Fanuc KAREL source: kt00120.KL

-- PROVISIONAL review KL for V770-1; original PC SHA256 89c0cbe0fdb6aaab56bf269acc3bfb9269b738d73fb216a7128dd25fbaf1ecd8
-- Incomplete behavior may be omitted. Consult companion uncertainty JSON. Do not deploy.
PROGRAM KT00120
%NOLOCKGROUP
VAR
  OUT : REAL
-- UNRESOLVED_DECL Y1 type=002018
-- UNRESOLVED_DECL H2 type=002017
BEGIN
  -- UNRESOLVED_PC offsets 5-19; opcodes 2E,22,9D,33,B2
  -- UNRESOLVED_PC offsets 24-38; opcodes 2E,22,9D,33,B4
  -- UNRESOLVED_PC offsets 43-72; opcodes 22,9D,33,B1,22,9D,33,B3,64,29,64,29,6C,23
  -- UNRESOLVED_PC offsets 77-81; opcodes 7F
END KT00120
